SUBAPPLICATION INI_OPC_PARAM_AX (* OPC_UA Parameter lesen/Schreiben, remanent per INI, mit AX-Ausgang fuer den gespeicherten Wert (z.B. Richtung). *)
  (* Standard: 61499-2; Description: Copyright (c) 2026 HR Agrartechnik GmbH This program and the accompanying materials are made available under the terms of the Eclipse Public License 2.0 which is available at https://www.eclipse.org/legal/epl-2.0/ SPDX-License-Identifier: EPL-2.0 *)
  (* Version 1.0, 2026-08-26, Franz Höpfinger, HR Agrartechnik GmbH, INI_OPC_PARAM_AR mit AX statt AR - initial API and implementation *)
  PACKAGE MyLib::sys;
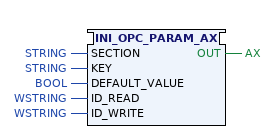
  VAR_INPUT
    SECTION : STRING; (* INI-Abschnitt (settings.ini) *)
    KEY : STRING; (* INI-Schluessel innerhalb SECTION *)
    DEFAULT_VALUE : BOOL; (* Wert falls in settings.ini nicht vorhanden *)
    ID_READ : WSTRING; (* OPC-UA-Verbindungsstring (READ) - Client schreibt hier einen neuen Wert *)
    ID_WRITE : WSTRING; (* OPC-UA-Verbindungsstring (WRITE) - aktuell gespeicherter Wert wird hier publiziert *)
  END_VAR
  PLUGS
    OUT : adapter::types::unidirectional::AX; (* Aktuell gespeicherter/geladener Wert *)
  END_PLUGS
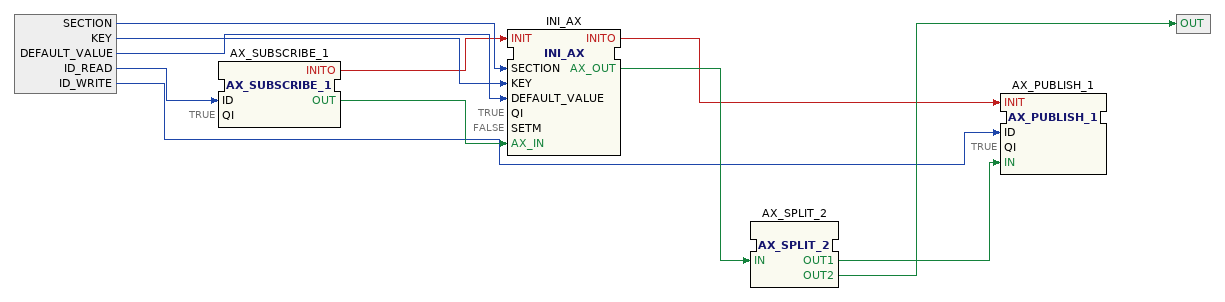
  FBS
    AX_SUBSCRIBE_1 : adapter::net::AX_SUBSCRIBE_1(QI := TRUE);
    AX_PUBLISH_1 : adapter::net::AX_PUBLISH_1(QI := TRUE);
    INI_AX : eclipse4diac::storage::INI_AX(QI := TRUE, SETM := FALSE);
    AX_SPLIT_2 : adapter::events::unidirectional::AX_SPLIT_2;
  END_FBS
  EVENT_CONNECTIONS
    AX_SUBSCRIBE_1.INITO TO INI_AX.INIT;
    INI_AX.INITO TO AX_PUBLISH_1.INIT;
  END_CONNECTIONS
  DATA_CONNECTIONS
    SECTION TO INI_AX.SECTION;
    KEY TO INI_AX.KEY;
    DEFAULT_VALUE TO INI_AX.DEFAULT_VALUE;
    ID_READ TO AX_SUBSCRIBE_1.ID;
    ID_WRITE TO AX_PUBLISH_1.ID;
  END_CONNECTIONS
  ADAPTER_CONNECTIONS
    AX_SUBSCRIBE_1.OUT TO INI_AX.AX_IN;
    AX_SPLIT_2.OUT1 TO AX_PUBLISH_1.IN;
    AX_SPLIT_2.OUT2 TO OUT;
    INI_AX.AX_OUT TO AX_SPLIT_2.IN;
  END_CONNECTIONS
END_SUBAPPLICATION
